# EPICS substitutions: modules/SAI/db/SAI_8MotorStatus.substitutions
file /opt/epics/modules/SAI/db/SAI_8MotorStatus.db {
    pattern {	ASYNPORT,	TMOT,		SCAN,		P,	R}
        { 	"pmac",		"1",		".2 second",	"FMB",	"MCTR01"}
}
